% RSLogix 500 project LAB2_BD_2.RSS, saved by version 8.40.00.08 %
PROJECT "UNTITLED"    % processor: SLC 500, 1747-L541 %

PROGRAM FILES
  LAD 2   37 rungs

DATA FILES
  O0 OUTPUT  68 elements
  I1 INPUT  68 elements
  S2 STATUS  164 elements
  B3 BINARY  3 elements
  T4 TIMER  34 elements
  C5 COUNTER  35 elements
  R6 CONTROL  1 elements
  N7 INTEGER  1 elements
  F8 FLOAT  1 elements

LADDER 2
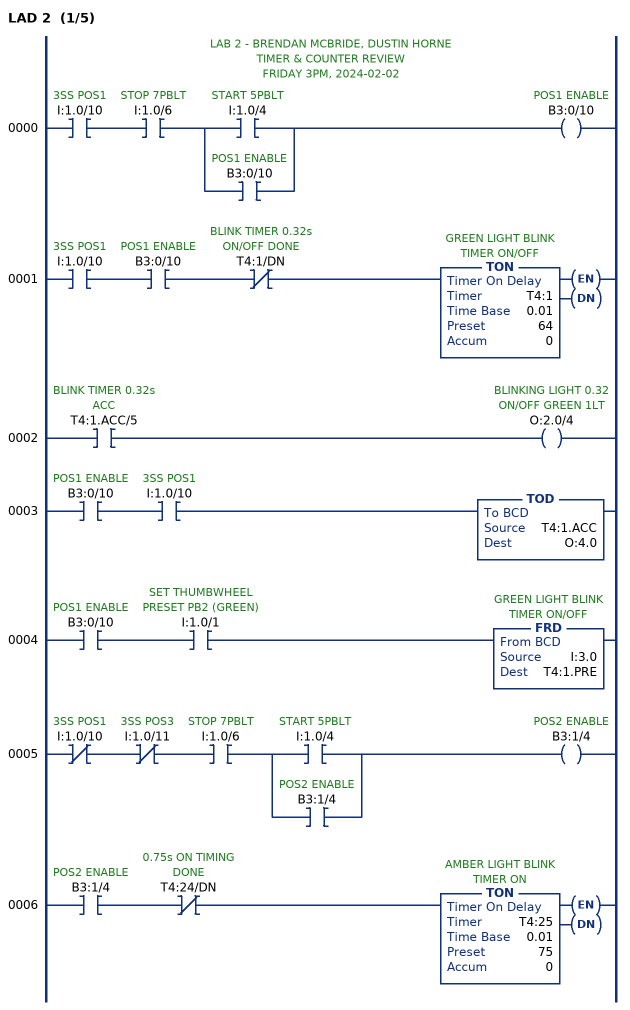
% Rung: 0 %
% LAB 2 - BRENDAN MCBRIDE, DUSTIN HORNE
% TIMER & COUNTER REVIEW
% FRIDAY 3PM, 2024-02-02 %
SOR XIC I:1.0/10 XIC I:1.0/6 BST XIC I:1.0/4 NXB XIC B3:0/10 BND OTE B3:0/10 EOR
%   I:1.0/10  "3SS POS1" %
%   I:1.0/6  "STOP 7PBLT" %
%   I:1.0/4  "START 5PBLT" %
%   B3:0/10  "POS1 ENABLE" %
% Rung: 1 %
SOR XIC I:1.0/10 XIC B3:0/10 XIO T4:1/DN TON T4:1 0.01 64 0 EOR
%   I:1.0/10  "3SS POS1" %
%   B3:0/10  "POS1 ENABLE" %
%   T4:1/DN  "BLINK TIMER 0.32s ON/OFF DONE" %
%   T4:1  "GREEN LIGHT BLINK TIMER ON/OFF" %
% Rung: 2 %
SOR XIC T4:1.ACC/5 OTE O:2.0/4 EOR
%   T4:1.ACC/5  "BLINK TIMER 0.32s ACC" %
%   O:2.0/4  "BLINKING LIGHT 0.32 ON/OFF GREEN 1LT" %
% Rung: 3 %
SOR XIC B3:0/10 XIC I:1.0/10 TOD T4:1.ACC O:4.0 EOR
%   B3:0/10  "POS1 ENABLE" %
%   I:1.0/10  "3SS POS1" %
%   T4:1  "GREEN LIGHT BLINK TIMER ON/OFF" %
% Rung: 4 %
SOR XIC B3:0/10 XIC I:1.0/1 FRD I:3.0 T4:1.PRE EOR
%   B3:0/10  "POS1 ENABLE" %
%   I:1.0/1  "SET THUMBWHEEL PRESET PB2 (GREEN)" %
%   T4:1  "GREEN LIGHT BLINK TIMER ON/OFF" %
% Rung: 5 %
SOR XIO I:1.0/10 XIO I:1.0/11 XIC I:1.0/6 BST XIC I:1.0/4 NXB XIC B3:1/4 BND OTE B3:1/4 EOR
%   I:1.0/10  "3SS POS1" %
%   I:1.0/11  "3SS POS3" %
%   I:1.0/6  "STOP 7PBLT" %
%   I:1.0/4  "START 5PBLT" %
%   B3:1/4  "POS2 ENABLE" %
% Rung: 6 %
SOR XIC B3:1/4 XIO T4:24/DN TON T4:25 0.01 75 0 EOR
%   B3:1/4  "POS2 ENABLE" %
%   T4:24/DN  "0.75s ON TIMING DONE" %
%   T4:25  "AMBER LIGHT BLINK TIMER ON" %

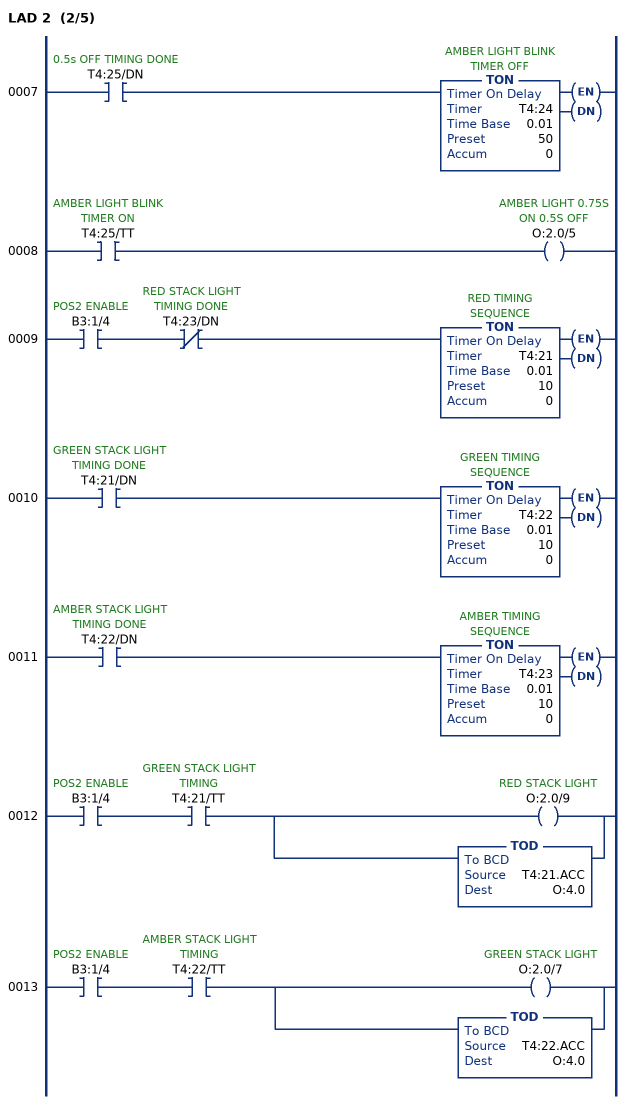
% Rung: 7 %
SOR XIC T4:25/DN TON T4:24 0.01 50 0 EOR
%   T4:25/DN  "0.5s OFF TIMING DONE" %
%   T4:24  "AMBER LIGHT BLINK TIMER OFF" %
% Rung: 8 %
SOR XIC T4:25/TT OTE O:2.0/5 EOR
%   T4:25  "AMBER LIGHT BLINK TIMER ON" %
%   O:2.0/5  "AMBER LIGHT 0.75S ON 0.5S OFF" %
% Rung: 9 %
SOR XIC B3:1/4 XIO T4:23/DN TON T4:21 0.01 10 0 EOR
%   B3:1/4  "POS2 ENABLE" %
%   T4:23/DN  "RED STACK LIGHT TIMING DONE" %
%   T4:21  "RED TIMING SEQUENCE" %
% Rung: 10 %
SOR XIC T4:21/DN TON T4:22 0.01 10 0 EOR
%   T4:21/DN  "GREEN STACK LIGHT TIMING DONE" %
%   T4:22  "GREEN TIMING SEQUENCE" %
% Rung: 11 %
SOR XIC T4:22/DN TON T4:23 0.01 10 0 EOR
%   T4:22/DN  "AMBER STACK LIGHT TIMING DONE" %
%   T4:23  "AMBER TIMING SEQUENCE" %
% Rung: 12 %
SOR XIC B3:1/4 XIC T4:21/TT BST OTE O:2.0/9 NXB TOD T4:21.ACC O:4.0 BND EOR
%   B3:1/4  "POS2 ENABLE" %
%   T4:21/TT  "GREEN STACK LIGHT TIMING" %
%   O:2.0/9  "RED STACK LIGHT" %
%   T4:21  "RED TIMING SEQUENCE" %
% Rung: 13 %
SOR XIC B3:1/4 XIC T4:22/TT BST OTE O:2.0/7 NXB TOD T4:22.ACC O:4.0 BND EOR
%   B3:1/4  "POS2 ENABLE" %
%   T4:22/TT  "AMBER STACK LIGHT TIMING" %
%   O:2.0/7  "GREEN STACK LIGHT" %
%   T4:22  "GREEN TIMING SEQUENCE" %

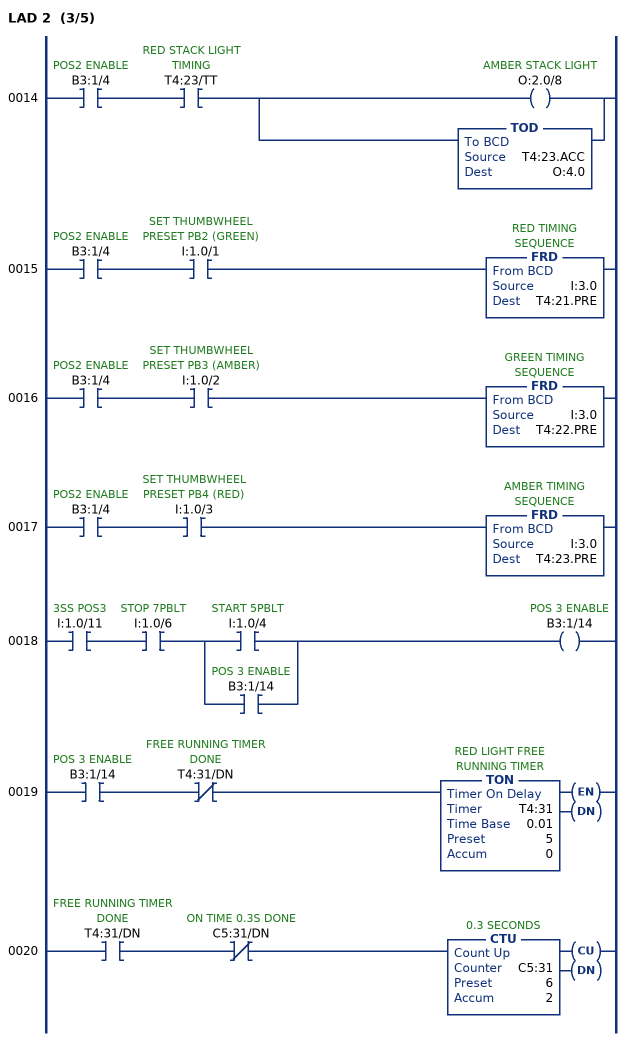
% Rung: 14 %
SOR XIC B3:1/4 XIC T4:23/TT BST OTE O:2.0/8 NXB TOD T4:23.ACC O:4.0 BND EOR
%   B3:1/4  "POS2 ENABLE" %
%   T4:23/TT  "RED STACK LIGHT TIMING" %
%   O:2.0/8  "AMBER STACK LIGHT" %
%   T4:23  "AMBER TIMING SEQUENCE" %
% Rung: 15 %
SOR XIC B3:1/4 XIC I:1.0/1 FRD I:3.0 T4:21.PRE EOR
%   B3:1/4  "POS2 ENABLE" %
%   I:1.0/1  "SET THUMBWHEEL PRESET PB2 (GREEN)" %
%   T4:21  "RED TIMING SEQUENCE" %
% Rung: 16 %
SOR XIC B3:1/4 XIC I:1.0/2 FRD I:3.0 T4:22.PRE EOR
%   B3:1/4  "POS2 ENABLE" %
%   I:1.0/2  "SET THUMBWHEEL PRESET PB3 (AMBER)" %
%   T4:22  "GREEN TIMING SEQUENCE" %
% Rung: 17 %
SOR XIC B3:1/4 XIC I:1.0/3 FRD I:3.0 T4:23.PRE EOR
%   B3:1/4  "POS2 ENABLE" %
%   I:1.0/3  "SET THUMBWHEEL PRESET PB4 (RED)" %
%   T4:23  "AMBER TIMING SEQUENCE" %
% Rung: 18 %
SOR XIC I:1.0/11 XIC I:1.0/6 BST XIC I:1.0/4 NXB XIC B3:1/14 BND OTE B3:1/14 EOR
%   I:1.0/11  "3SS POS3" %
%   I:1.0/6  "STOP 7PBLT" %
%   I:1.0/4  "START 5PBLT" %
%   B3:1/14  "POS 3 ENABLE" %
% Rung: 19 %
SOR XIC B3:1/14 XIO T4:31/DN TON T4:31 0.01 5 0 EOR
%   B3:1/14  "POS 3 ENABLE" %
%   T4:31/DN  "FREE RUNNING TIMER DONE" %
%   T4:31  "RED LIGHT FREE RUNNING TIMER" %
% Rung: 20 %
SOR XIC T4:31/DN XIO C5:31/DN CTU C5:31 6 2 EOR
%   T4:31/DN  "FREE RUNNING TIMER DONE" %
%   C5:31/DN  "ON TIME 0.3S DONE" %
%   C5:31  "0.3 SECONDS" %

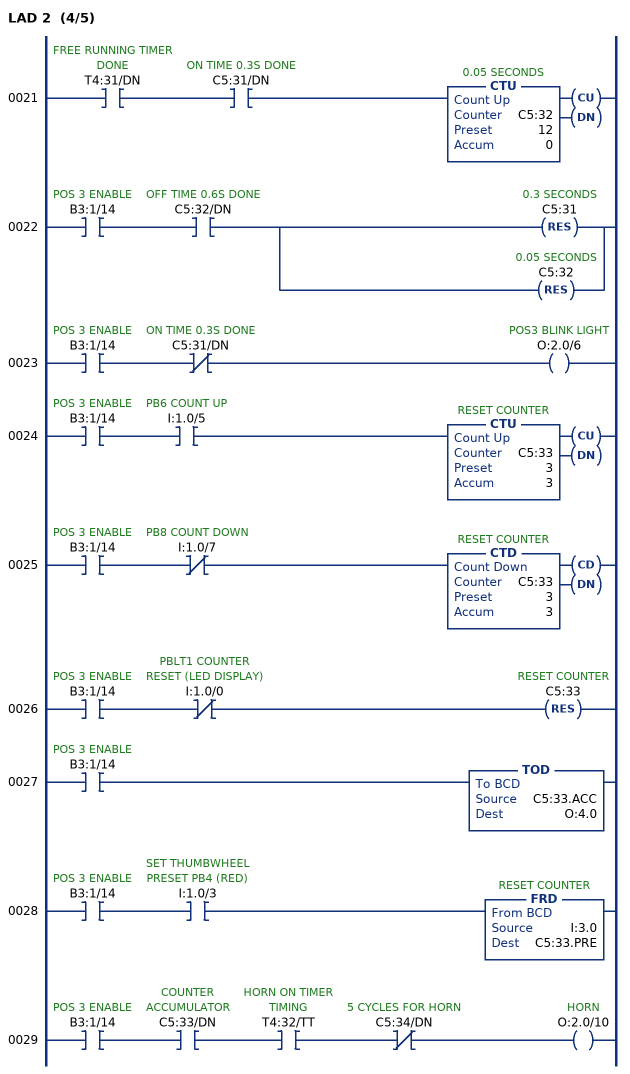
% Rung: 21 %
SOR XIC T4:31/DN XIC C5:31/DN CTU C5:32 12 0 EOR
%   T4:31/DN  "FREE RUNNING TIMER DONE" %
%   C5:31/DN  "ON TIME 0.3S DONE" %
%   C5:32  "0.05 SECONDS" %
% Rung: 22 %
SOR XIC B3:1/14 XIC C5:32/DN BST RES C5:31 NXB RES C5:32 BND EOR
%   B3:1/14  "POS 3 ENABLE" %
%   C5:32/DN  "OFF TIME 0.6S DONE" %
%   C5:31  "0.3 SECONDS" %
%   C5:32  "0.05 SECONDS" %
% Rung: 23 %
SOR XIC B3:1/14 XIO C5:31/DN OTE O:2.0/6 EOR
%   B3:1/14  "POS 3 ENABLE" %
%   C5:31/DN  "ON TIME 0.3S DONE" %
%   O:2.0/6  "POS3 BLINK LIGHT" %
% Rung: 24 %
SOR XIC B3:1/14 XIC I:1.0/5 CTU C5:33 3 3 EOR
%   B3:1/14  "POS 3 ENABLE" %
%   I:1.0/5  "PB6 COUNT UP" %
%   C5:33  "RESET COUNTER" %
% Rung: 25 %
SOR XIC B3:1/14 XIO I:1.0/7 CTD C5:33 3 3 EOR
%   B3:1/14  "POS 3 ENABLE" %
%   I:1.0/7  "PB8 COUNT DOWN" %
%   C5:33  "RESET COUNTER" %
% Rung: 26 %
SOR XIC B3:1/14 XIO I:1.0/0 RES C5:33 EOR
%   B3:1/14  "POS 3 ENABLE" %
%   I:1.0/0  "PBLT1 COUNTER RESET (LED DISPLAY)" %
%   C5:33  "RESET COUNTER" %
% Rung: 27 %
SOR XIC B3:1/14 TOD C5:33.ACC O:4.0 EOR
%   B3:1/14  "POS 3 ENABLE" %
%   C5:33  "RESET COUNTER" %
% Rung: 28 %
SOR XIC B3:1/14 XIC I:1.0/3 FRD I:3.0 C5:33.PRE EOR
%   B3:1/14  "POS 3 ENABLE" %
%   I:1.0/3  "SET THUMBWHEEL PRESET PB4 (RED)" %
%   C5:33  "RESET COUNTER" %
% Rung: 29 %
SOR XIC B3:1/14 XIC C5:33/DN XIC T4:32/TT XIO C5:34/DN OTE O:2.0/10 EOR
%   B3:1/14  "POS 3 ENABLE" %
%   C5:33/DN  "COUNTER ACCUMULATOR" %
%   T4:32/TT  "HORN ON TIMER TIMING" %
%   C5:34/DN  "5 CYCLES FOR HORN" %
%   O:2.0/10  "HORN" %

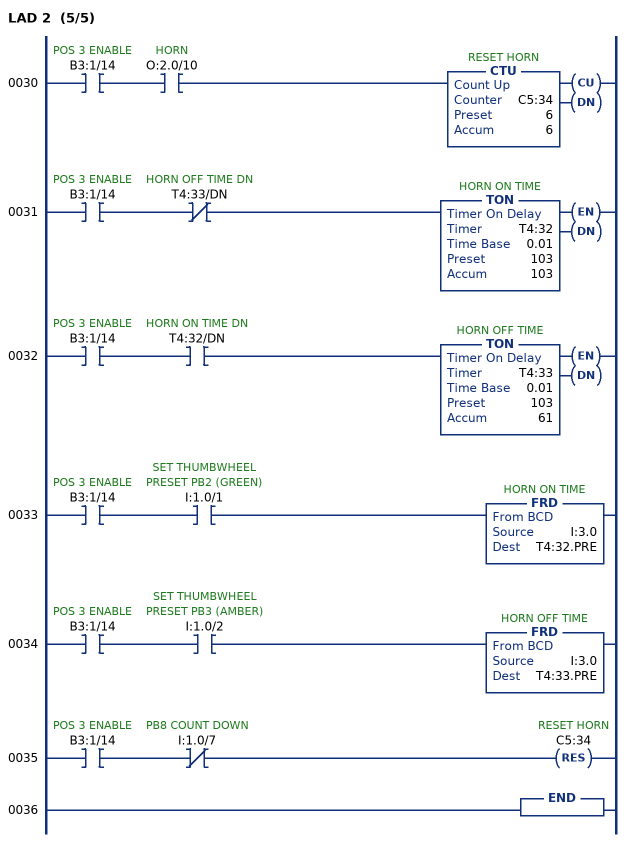
% Rung: 30 %
SOR XIC B3:1/14 XIC O:2.0/10 CTU C5:34 6 6 EOR
%   B3:1/14  "POS 3 ENABLE" %
%   O:2.0/10  "HORN" %
%   C5:34  "RESET HORN" %
% Rung: 31 %
SOR XIC B3:1/14 XIO T4:33/DN TON T4:32 0.01 103 103 EOR
%   B3:1/14  "POS 3 ENABLE" %
%   T4:33/DN  "HORN OFF TIME DN" %
%   T4:32  "HORN ON TIME" %
% Rung: 32 %
SOR XIC B3:1/14 XIC T4:32/DN TON T4:33 0.01 103 61 EOR
%   B3:1/14  "POS 3 ENABLE" %
%   T4:32/DN  "HORN ON TIME DN" %
%   T4:33  "HORN OFF TIME" %
% Rung: 33 %
SOR XIC B3:1/14 XIC I:1.0/1 FRD I:3.0 T4:32.PRE EOR
%   B3:1/14  "POS 3 ENABLE" %
%   I:1.0/1  "SET THUMBWHEEL PRESET PB2 (GREEN)" %
%   T4:32  "HORN ON TIME" %
% Rung: 34 %
SOR XIC B3:1/14 XIC I:1.0/2 FRD I:3.0 T4:33.PRE EOR
%   B3:1/14  "POS 3 ENABLE" %
%   I:1.0/2  "SET THUMBWHEEL PRESET PB3 (AMBER)" %
%   T4:33  "HORN OFF TIME" %
% Rung: 35 %
SOR XIC B3:1/14 XIO I:1.0/7 RES C5:34 EOR
%   B3:1/14  "POS 3 ENABLE" %
%   I:1.0/7  "PB8 COUNT DOWN" %
%   C5:34  "RESET HORN" %
% Rung: 36 %
SOR END EOR

OTHER DOCUMENTED ADDRESSES
  C5:34.ACC  "HORN COUNTER ACC >= PRESET"
  I:0.0/8  "THUMBWHEEL PRESET ADJUST"

DATA TABLE (non-zero values as saved)
DATA B3
% B3:0 % 0X0000 0X4000 0X0000
DATA T4
% .PRE .ACC %
% T4:1 % 64 0
% T4:21 % 10 0
% T4:22 % 10 0
% T4:23 % 10 0
% T4:24 % 50 0
% T4:25 % 75 0
% T4:31 % 5 0
% T4:32 % 103 103
% T4:33 % 103 61
DATA C5
% .PRE .ACC %
% C5:31 % 6 2
% C5:32 % 12 0
% C5:33 % 3 3
% C5:34 % 6 6
